FUNCTION_BLOCK T_ModeChangeFromProductionToMaintenance EXTENDS T_UnitTestBase
VAR
  mockState : T_MockStateModule;
  modeManager : T_ModeManager(mockState);
  expected, actual : UINT;
END_VAR

CycleModuleLogicToAllowChangesToFilterThrough();
modeManager.ChangeMode(E_PMLUnitMode.ePMLUnitMode_Maintenance);
CycleModuleLogicToAllowChangesToFilterThrough();

actual := TO_UINT(modeManager.CurrentMode);
expected := TO_UINT(E_PMLUnitMode.ePMLUnitMode_Maintenance);
assertion.AssertEquals_UINT(expected, actual, 'actual := TO_UINT(modeManager.CurrentMode)');
TestFinished();

METHOD CycleModuleLogicToAllowChangesToFilterThrough : BOOL
VAR_INST
	i: INT;

END_VAR
FOR i := 0 TO 25 DO
  modeManager.CyclicLogic();
END_FOR
END_METHOD

END_FUNCTION_BLOCK

(* stored: Version 1.1.0.1, ProductVersion 3.1.4024.12
   POU T_ModeChangeFromProductionToMaintenance: Id {738a0f00-8349-4471-bf75-f1cc1179c765}, SpecialFunc None
   Method CycleModuleLogicToAllowChangesToFilterThrough: Id {77dca678-9999-44f8-ba35-3484f59b06bc} *)
